Fanuc KAREL source: VT_CLR_QUEUE.kl

PROGRAM T
%NOLOCKGROUP
VAR
 v0 : INTEGER
 v1 : INTEGER
BEGIN
 VT_CLR_QUEUE(v0, v1)
END T
